// TwinCAT 3 PLC project PLC
// ProgramVersion: 3.1.4024.0
// libraries:
//   Tc2_Standard, * (Beckhoff Automation GmbH)
//   Tc2_System, * (Beckhoff Automation GmbH)
//   Tc3_Module, * (Beckhoff Automation GmbH)
// project tree:
//   GVLs/ GVL.TcGVL
//   / PlcTask.TcTTO
//   POUs/ FillBox.TcPOU, MAIN.TcPOU, StartStop.TcPOU, Vision.TcPOU
// real-time tasks:
//   TASK PlcTask: cycle T#10ms, priority 20, ADS port 350

CONFIGURATION PLC
    RESOURCE PLC ON TwinCAT3
        TASK PlcTask(INTERVAL := T#10ms, PRIORITY := 20);
        PROGRAM MAIN WITH PlcTask : MAIN;
    END_RESOURCE
END_CONFIGURATION

// ---- GVLs/GVL.TcGVL
{attribute 'qualified_only'}
VAR_GLOBAL
		RunBit			:	BOOL;		// internal control bit. Plant running if TRUE
		K3Flag			:	BOOL:=TRUE;	// control the K5 cylinder. True if cylinder is up
END_VAR

// ---- POUs/MAIN.TcPOU
PROGRAM MAIN
VAR
END_VAR

FillBox();
Vision();
StartStop();

END_PROGRAM

// ---- POUs/FillBox.TcPOU
PROGRAM FillBox
VAR
		BoxCylinder				:	BOOL; 	// cylinder to stop box to be filled
		ItemReady				:	BOOL;	// item ready to be moved to the box by the robot
		StartRobotPrg			:	BOOL;	// start robot program
		RobotMoveOneItem		:	BOOL;	// signal to robot: move one item
		BoxReadyToFill			:	BOOL;	// a box is ready to be filled
		RobotMovedAllItems		: 	BOOL;	// signal from robot. Robot has moved all items
END_VAR
VAR // added by the converter: edge detectors and wires of the graphical bodies
    _w1 : BOOL;
END_VAR

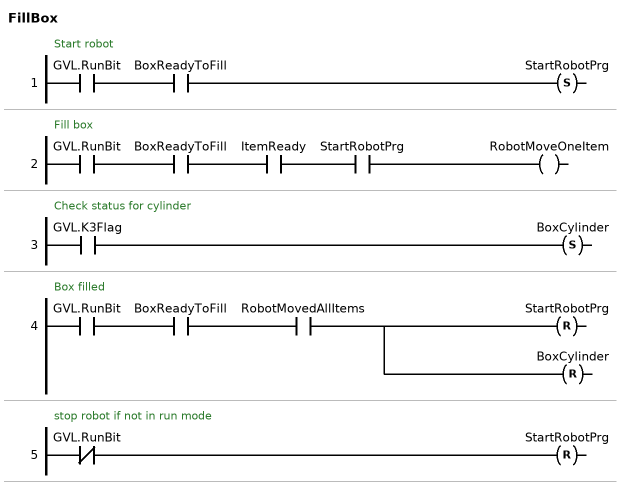
// NETWORK 1
// Start robot
StartRobotPrg S= GVL.RunBit AND BoxReadyToFill;

// NETWORK 2
// Fill box
RobotMoveOneItem := GVL.RunBit AND BoxReadyToFill AND ItemReady AND StartRobotPrg;

// NETWORK 3
// Check status for cylinder
BoxCylinder S= GVL.K3Flag;

// NETWORK 4
// Box filled
_w1 := GVL.RunBit AND BoxReadyToFill AND RobotMovedAllItems;
StartRobotPrg R= _w1;
BoxCylinder R= _w1;

// NETWORK 5
// stop robot if not in run mode
StartRobotPrg R= NOT GVL.RunBit;

END_PROGRAM

// ---- POUs/Vision.TcPOU
PROGRAM Vision
VAR
		BoxLeavesArea	:	BOOL;	// box leaves the filling area and is on the way to vision check
		BoxReadyVision	:	BOOL;	// box ready for vision check
		VisionCheckOk	:	BOOL;	// signal from vision. TRUE if box is OK
		LampBoxOk		:	BOOL;	// signal lamp. Box OK
		LampBoxNok		:	BOOL;	// signal lamp. Box NOK
		StartVision		:	BOOL;	// start vision check
END_VAR
VAR // added by the converter: edge detectors and wires of the graphical bodies
    _w1, _w2 : BOOL;
END_VAR

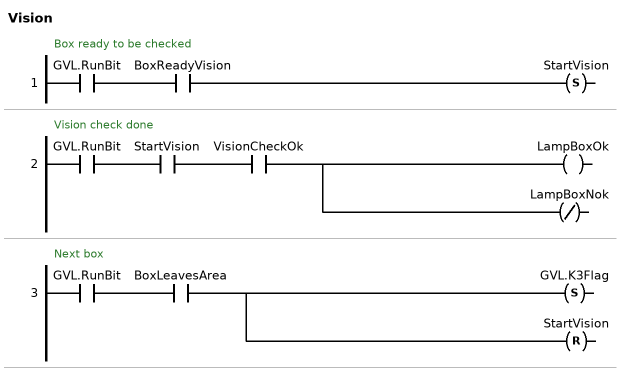
// NETWORK 1
// Box ready to be checked
StartVision S= GVL.RunBit AND BoxReadyVision;

// NETWORK 2
// Vision check done
_w1 := GVL.RunBit AND StartVision AND VisionCheckOk;
LampBoxOk := _w1;
LampBoxNok := NOT _w1;

// NETWORK 3
// Next box
_w2 := GVL.RunBit AND BoxLeavesArea;
GVL.K3Flag S= _w2;
StartVision R= _w2;

END_PROGRAM

// ---- POUs/StartStop.TcPOU
PROGRAM StartStop
VAR
	StartPb			:	BOOL;	// start switch (NO)
	StopPb			:	BOOL;	// stop switch (NC)
	Motor1			:	BOOL;	// run conveyor 1 belt
	Motor2			:	BOOL;	// run conveyor 2 belt	
END_VAR
VAR // added by the converter: edge detectors and wires of the graphical bodies
    _w1 : BOOL;
END_VAR

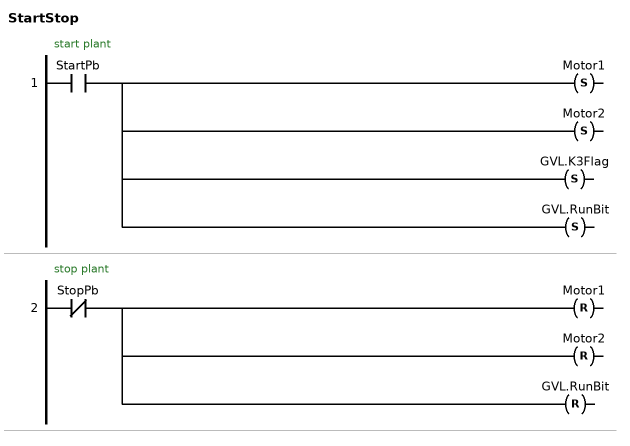
// NETWORK 1
// start plant
Motor1 S= StartPb;
Motor2 S= StartPb;
GVL.K3Flag S= StartPb;
GVL.RunBit S= StartPb;

// NETWORK 2
// stop plant
_w1 := NOT StopPb;
Motor1 R= _w1;
Motor2 R= _w1;
GVL.RunBit R= _w1;

END_PROGRAM
